FUNCTION_BLOCK E_CYCLE (* Periodic(cyclic)Generation of an Event *)
  (* Standard: 61499-1; Classification: Event Processing; Function: Cyclic Event Generation *)
  (* Version 0.2, 2006-04-18, JHC, Holobloc Inc, Added resource-side primitives. *)
  (* Version 0.1, 2002-01-30, JHC, Rockwell Automation, Changed from basic to SIFB, added change_DT functionality. *)
  (* Version 0.0, 2001-04-14, JHC, Rockwell Automation, First XML version. *)
  (* Compiler header: package fb.rt.events; *)
  (* Compiler Java Sun JDK 1.5.0 *)
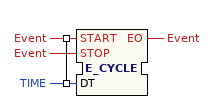
  EVENT_INPUT
    START WITH DT;
    STOP;
  END_EVENT
  EVENT_OUTPUT
    EO; (* Periodic event at period DT,starting at DT after START *)
  END_EVENT
  VAR_INPUT
    DT : TIME; (* Period between events *)
  END_VAR
  SERVICE E_CYCLE/resource
    SEQUENCE event_cycle
      E_CYCLE.START(DT) -> resource.start_cycling(DT);
      resource.timeout() -> E_CYCLE.EO();
      resource.timeout() -> E_CYCLE.EO();
      resource.timeout() -> E_CYCLE.EO();
    END_SEQUENCE
    SEQUENCE cycle_canceled
      E_CYCLE.START(DT) -> resource.start_cycling(DT);
      resource.timeout() -> E_CYCLE.EO();
      E_CYCLE.STOP() -> resource.stop_cycling();
    END_SEQUENCE
  END_SERVICE
END_FUNCTION_BLOCK
